// ---- POUs/UserPOUs/UserFunctions/ToRobotPoseSimple.TcPOU
FUNCTION ToRobotPoseSimple
VAR_INPUT
	x, y, theta : LREAL;
END_VAR
VAR
END_VAR
VAR_OUTPUT
	RobotPose : RobotPoseSimple;
END_VAR

RobotPose.x := x;
RobotPose.y := y;
RobotPose.theta := theta;

END_FUNCTION

// ---- POUs/UserPOUs/TrajectoryControl.TcPOU
//TrajectoryControl:
//GW2 side of the interface to GW3
FUNCTION_BLOCK TrajectoryControl
VAR_INPUT
	//interface to GW3
	// INPUTS to GW3
	xBoEnable AT%Q*: BOOL := FALSE;							// Freigabesignal für Fahrt, Roboter stoppt bei FALSE
	waypointList AT%Q*: ARRAY[0..100] OF RobotPoseSimple;	// Wegpunktliste mit Roboter-Posen in globalen Koordinaten (x, y, theta)
	newWaypointListAvailable AT%Q*: BOOL := FALSE;			// Status-Bit zur Signalisierung einer neuen WP-Liste
	xBoReset  AT%Q*: BOOL := FALSE;							
END_VAR
VAR_OUTPUT
	// OUTPUTS from GW3		
	yBoArrivedAtDestination AT%I*: BOOL 			:= FALSE;	// TRUE, wenn Ziel erreicht, Ziel entspricht letzten gültigen WP
	yUintWaypointIndex  	AT%I*: INT 				:= 0;		// COUNTER zur Anzeige, des Indexes des nächstes WP
	yRPposition 			AT%I*: RobotPoseSimple;				// aktuelle Roboterposition, für Simulationszwecke;
	yControllerState   	 	AT%I*: ControllerState;
	yVworldRef				AT%I*: RobotPoseSimple;
END_VAR

METHOD setWaypointList : BOOL
VAR_INPUT
	newWaypointList : ARRAY [0..100] OF RobotPoseSimple;
END_VAR
waypointList := newWaypointList;
END_METHOD

END_FUNCTION_BLOCK

// ---- POUs/UserPOUs/UserFunctions/ZEROS_RobotPoseSimple.TcPOU
FUNCTION ZEROS_RobotPoseSimple : Array[0..100] OF RobotPoseSimple
VAR_IN_OUT
	arr: ARRAY [0..100] OF RobotPoseSimple;
END_VAR
VAR
	i: INT;
END_VAR

FOR i := 0 TO 100 BY 1 DO
	arr[i] := ToRobotPoseSimple(x := 0, y := 0, theta := 0);
END_FOR

END_FUNCTION

// ---- POUs/UserPOUs/GW2/DS_GW1.TcPOU
PROGRAM DS_GW1
VAR
// Identifikation des Roboters
    //Robot_Number	AT%I*	: INT;	

// Local Variables for Mqtt Client handling
	fbIotMqttClient : FB_IotMqttClient;
	//ClientId : STRING(255);
    //ClientId : STRING(255) := CONCAT('HAWino_', INT_TO_STRING(.Var_HAWIno.Robot_Number));
	bSetParameter 	: BOOL := TRUE;
	bConnect 		: BOOL := TRUE;	
	
// Publish message
	initMQTT : BOOL := FALSE;
	sTopicPubToPowerMgmt : STRING(255); //:= CONCAT('Robots/PowerMgmt/Robot_', INT_TO_STRING(.Var_HAWIno.Robot_Number)); 	// ToDo: Bisher ist die Nummer des HAWino fest kodiert
	sTopicPubToPowerMgmt_SOC : STRING(255);// := CONCAT('Robots/PowerMgmt/SoC_Robot_', INT_TO_STRING(.Var_HAWIno.Robot_Number)); 
	sPayloadPub : STRING(2000);
	sPayloadPub1 : STRING(2000);		
	fbTimerPub 	: TON := (PT:=T#500MS);									// Intervall für das Senden des Akku-Status
	
//Received message
	bSubscribed    : BOOL;
	sTopicSubToPowerMgmt : STRING(255);// := CONCAT('PowerMgmt/Robots/Robot_', INT_TO_STRING(.Var_HAWIno.Robot_Number));	// ToDo: Bisher ist die Nummer des HAWino fest kodiert
	sTopicRcv      : STRING(255);
	sPayloadRcv    : STRING(255);
	fbMessageQueue : FB_IotMqttMessageQueue;
    fbMessage      : FB_IotMqttMessage;
	hrErrorOccurred : HRESULT; 			// Enthlt dern letzten augetretenen Fehler
	
	//wir geändert
	//sTopicSubToGW1: STRING(255);
	
// Variables for JSON
	fbJson			: FB_JsonSaxWriter;
	fbJsonDataType 	: FB_JsonReadWriteDataType;
	sJsonDoc       	: STRING(2000); 
	
// Local Variables for TwinCAT IoT Communication (TF6701) with direct link to EK1200 and TcCom
	//stMqtt_HAWino_In	AT%I*	: ST_PwrMgmt_HAWino_In;		// Attention! Don't link TIME Variables, otherwise we get an error!
	//stMqtt_HAWino_Out	AT%Q*	: ST_PwrMgmt_HAWino_Out;
	
	stMqtt_HAWino_In	 AT%I*: ST_PwrMgmt_HAWino_In;		// Attention! Don't link TIME Variables, otherwise we get an error!
	stMqtt_HAWino_Out	 AT%Q*: ST_PwrMgmt_HAWino_Out;
	
	SOC_Out : STRING(255);
	nBatteryTemperature	AT%I*	: INT;
	
	bComCheckAnswer	AT%Q*	: BOOL;
	
	stMqtt_HAWinoValues	: ST_PwrMgmt_HAWino;
	
	
// Timer to create a time stamp
	fbTimerTimestamp : TON := (PT:=T#71582M47S295MS);
	
// Local Vaiables to evaluate and act to input
	fbComCheckFlag	: RS;
	
	
	
	sTopicSubToFleetMgmt: STRING;
	Reset1: BOOL;
	//Input synccheck. robotdata has been read and can be used.
	txtReadInit AT%I* : BOOL := FALSE;
	
	// eigene Variablen	
	feedback: ARRAY[0..7] OF STRING := ['Verfügbar', 'Auftrag angenommen', 'Auf Anfahrt', 'Teil aufgenommen', 
											'Abmeldung', 'Auf Transport', 'Anmeldung', 'Teil abgelegt'];
	sTopicPubToGW1: STRING(255) := CONCAT('VPJ/Robot_', INT_TO_STRING(.Var_HAWIno.Robot_Number));
	s0: BOOL := 1;
	s1, s2, s3, s4, s5, s6, s7: BOOL := 0;
	AuftragDa: BOOL;
	Timer1 : TON;
	Timer2 : TON;
	startTime1: BOOL;
	startTime2: BOOL;
	WerkstueckAusgelesen: BOOL;
	i: INT := 0;

END_VAR

//Dummy Programm als Schnittstelle für Gewerk 1

//Case machen! preop op
txtReadInit := MQTT.txtReadInit;
IF txtReadInit THEN
	IF NOT initMQTT THEN
		sTopicPubToPowerMgmt  := CONCAT('Robots/PowerMgmt/Robot_', INT_TO_STRING(.Var_HAWIno.Robot_Number)); 	
		sTopicPubToPowerMgmt_SOC  := CONCAT('Robots/PowerMgmt/SoC_Robot_', INT_TO_STRING(.Var_HAWIno.Robot_Number)); 
		sTopicSubToPowerMgmt  := CONCAT('PowerMgmt/Robots/Robot_', INT_TO_STRING(.Var_HAWIno.Robot_Number));
		//sTopicSubToGW1  := CONCAT('VPJ/Robot_', INT_TO_STRING(.Var_HAWIno.Robot_Number));
		initMQTT:= TRUE;
	END_IF
	
	stMqtt_HAWinoValues.Output.nRobotNumber := .Var_HAWIno.Robot_Number;			// Anpassen für jeden HAWino
	
	fbTimerTimestamp(In:= NOT fbTimerTimestamp.Q, ET=>stMqtt_HAWinoValues.Output.tTimestamp);
	
	stMqtt_HAWinoValues.Output.fSoC := stMqtt_HAWino_In.fSoC;
	
	stMqtt_HAWinoValues.Output.fActualBatteryCurrent := stMqtt_HAWino_In.fActualBatteryCurrent;
	stMqtt_HAWinoValues.Output.fActualBatteryVoltage := stMqtt_HAWino_In.fActualBatteryVoltage;
	
	//stMqtt_HAWinoValues.Output.fActualBatteryCurrent := stMqtt_HAWino_In.fActualBatteryCurrent;
	//stMqtt_HAWinoValues.Output.fActualBatteryVoltage := stMqtt_HAWino_In.fActualBatteryVoltage;
	
	
	
	
	// Skalierung der Temperaturwerte des Akkus
	stMqtt_HAWinoValues.Output.fBatteryTemperature := FKT_Scale(Rohwert := nBatteryTemperature, 
																	X1 := -500,
																	X2 := 1500, 
																	Y1 := -50,
																	Y2 := 150);
																	
	// Ausgabe der erwarteten Laufzeit des Roboters
	stMqtt_HAWinoValues.Output.nEstimatedRunningTime	:= LIMIT(0,stMqtt_HAWino_In.nEstimatedRunningTime,172800);		// Max. 48 Stunden sollen dargestellt werden
	stMqtt_HAWinoValues.Output.nEstimatedChargingTime	:= LIMIT(0,stMqtt_HAWino_In.nEstimatedChargingTime,172800);		// Max. 48 Stunden sollen dargestellt werden
	
	
	// Antworten auf den Kommunikationstest und des Ladetests
	stMqtt_HAWinoValues.Output.bCheckCurrentDetected := stMqtt_HAWino_In.bCheckCurrentDetected;
	stMqtt_HAWinoValues.Output.bComCheckAnswer := stMqtt_HAWino_In.bComCheckAnswer;
	
	
			
	
	
	
	
	//
	// Setting the parameters for establishing the connection to the Mqtt Broker and initializing the connection.
	//
	IF bSetParameter THEN
		fbIotMqttClient.sHostName := '192.168.0.11';	// IP-Adresse des Servers
		fbIotMqttClient.nHostPort := 1883;
		//fbIotMqttClient.sClientId := ClientId;
		fbIotMqttClient.sClientId := CONCAT('Robot_', INT_TO_STRING(.Var_HAWIno.Robot_Number));
		fbIotMqttClient.sTopicPrefix := '';
		//fbIotMqttClient.nKeepAlive:= 60; 
		fbIotMqttClient.sUserName:= 'VPJ';
		fbIotMqttClient.sUserPassword:= 'R462';
		//fbIotMqttClient.stWill:= ; 
		//fbIotMqttClient.stTLS:= ;
		fbIotMqttClient.ipMessageQueue := fbMessageQueue;
	
		bSetParameter := FALSE;
	END_IF
	
	
	//
	// This method -> MUST BE CALLED CYCLICALLY <- to ensure background communication with the MQTT broker.
	//
	fbIotMqttClient.Execute(bConnect);
	
	IF fbIotMqttClient.bError THEN
		// ToDo: add error logging here
		hrErrorOccurred := fbIotMqttClient.hrErrorCode;
	END_IF
	
		
	IF fbIotMqttClient.bConnected THEN		// Kontrolle, ob der Broker verbunden ist
		IF NOT bSubscribed THEN
			//
			// Abbonieren der Toopics, welche vom PowerMgmt kommen
			//
			bSubscribed := fbIotMqttClient.Subscribe(sTopic:=sTopicSubToPowerMgmt, eQoS:=TcIotMqttQos.AtMostOnceDelivery);
			IF fbIotMqttClient.bError THEN
				// ToDo: add my error logging here
				hrErrorOccurred := fbIotMqttClient.hrErrorCode;
			END_IF
			
			//
			// Abbonieren der Toopics, welche vom Gewerk 1 kommen
			//
			//Abbonieren von Topic: VPJ/Roboter
			//bSubscribed := fbIotMqttClient.Subscribe(sTopic:=sTopicSubToGW1, eQoS:=TcIotMqttQos.AtMostOnceDelivery);
			
			
			//bSubscribed := fbIotMqttClient.Subscribe(sTopic:=sTopicSubToFleetMgmt, eQoS:=TcIotMqttQos.AtMostOnceDelivery);
			//IF fbIotMqttClient.bError THEN
				// ToDo: add my error logging here
			//	hrErrorOccurred := fbIotMqttClient.hrErrorCode;
			//END_IF
			
		END_IF
	END_IF	
	
	
	
	// Senden der MQTT- Nachrichten
	
	
	IF fbIotMqttClient.bConnected THEN			// Kontrolle, ob Broker verbunden ist
		fbTimerPub(IN:=TRUE);
		
		//
		// publish new paylod every 500 MS
		//
		IF fbTimerPub.Q THEN					// Abwarten des oben eingestellten Intervalls
			fbTimerPub(IN:=FALSE);
			
			//
			// Nachricht an PowerMgmt
			//
			fbJson.ResetDocument();
			fbJsonDataType.AddJsonValueFromSymbol(fbJson, 'ST_PwrMgmt_HAWino_In', SIZEOF(stMqtt_HAWinoValues.Output), ADR(stMqtt_HAWinoValues.Output));
			//sJsonDoc := fbJson.GetDocument();
			fbJson.CopyDocument(sJsonDoc, SIZEOF(sJsonDoc));
			
			sPayloadPub := sJsonDoc;	
			fbIotMqttClient.Publish(sTopic:= sTopicPubToPowerMgmt, 
										pPayload:= ADR(sPayloadPub), 
										nPayloadSize:= LEN2(ADR(sPayloadPub))+1, 										
										eQoS:= TcIotMqttQos.AtMostOnceDelivery, 
										bRetain:= FALSE, 
										bQueue:= FALSE);
									
			
			SOC_Out	:= CONCAT( '{"SoC" : ',LREAL_TO_STRING(stMqtt_HAWinoValues.Output.fSoC));
			SOC_Out	:= CONCAT( SOC_Out,'}');
			
			
			
			
			//SOC_Out := 	LREAL_TO_STRING(stMqtt_HAWinoValues.Output.fSoC);
			
						
			fbIotMqttClient.Publish(sTopic:= sTopicPubToPowerMgmt_SOC, 
										pPayload:=ADR(SOC_Out), 
										nPayloadSize:= INT_TO_UDINT(LEN(SOC_Out)),
										eQoS:= TcIotMqttQos.AtMostOnceDelivery, 
										bRetain:= FALSE, 
										bQueue:= FALSE);
										
										
			IF fbIotMqttClient.bError THEN
				// ToDo: add error logging here
				hrErrorOccurred := fbIotMqttClient.hrErrorCode;
			END_IF	
			
			//
			// ...
			//	
			//
			// Nachricht an GW1 - Produktionsauftrag
			//
			//Statemaschine
			Timer1(IN:= startTime1, PT:=T#10S);
			Timer2(IN:= startTime2, PT:=T#10S);
	
			//Rückmeldung Verfügbar
			sPayloadPub1 := CONCAT( '{"status" : ', feedback[i]);
			sPayloadPub1 := CONCAT( sPayloadPub1,'}');
			
			fbIotMqttClient.Publish(sTopic:= sTopicPubToGW1, 
											pPayload:=ADR(sPayloadPub1), 
											nPayloadSize:= INT_TO_UDINT(LEN(sPayloadPub1)),
											eQoS:= TcIotMqttQos.AtMostOnceDelivery, 
											bRetain:= FALSE, 
											bQueue:= FALSE);
											
			i := 2;
											
			//Warten auf Auftrag
			IF s0 AND NOT s1 AND AuftragDa THEN
				s0 := 0; s1 := 1;
				//Rückmeldung Auftrag angenommen
				i := 1;
				//fbIotMqttClient.Publish(sTopic:= sTopicPubToGW1, 
											//pPayload:=ADR(feedback[1]), 
											//nPayloadSize:= INT_TO_UDINT(LEN(feedback[1])),
											//eQoS:= TcIotMqttQos.AtMostOnceDelivery, 
											//bRetain:= FALSE, 
											//bQueue:= FALSE);
				startTime1 := 1;
			END_IF
			IF s1 AND NOT s2 AND Timer1.Q THEN
				startTime1 := 0;
				s1 := 0; s2 := 1;
				//Rückmeldung Auf Anfahrt
				i := 2;
				//fbIotMqttClient.Publish(sTopic:= sTopicPubToGW1, 
											//pPayload:=ADR(feedback[2]), 
											//nPayloadSize:= INT_TO_UDINT(LEN(feedback[2])),
											//eQoS:= TcIotMqttQos.AtMostOnceDelivery, 
											//bRetain:= FALSE, 
											//bQueue:= FALSE);
				startTime2 := 1;
			END_IF
			IF s2 AND NOT s3 AND Timer2.Q THEN
				startTime2 := 0;
				s2 := 0; s3 := 1;
				//Rückmeldung Teil aufgenommen
				i := 3;
				fbIotMqttClient.Publish(sTopic:= sTopicPubToGW1, 
											pPayload:=ADR(feedback[3]), 
											nPayloadSize:= INT_TO_UDINT(LEN(feedback[3])),
											eQoS:= TcIotMqttQos.AtMostOnceDelivery, 
											bRetain:= FALSE, 
											bQueue:= FALSE);
				startTime1 := 1;
			END_IF
			IF s3 AND NOT s4 AND Timer1.Q THEN
				startTime1 := 0;
				s3 := 0; s4 := 1;
				//Rückmeldung Abmeldung
				i := 4;
				//fbIotMqttClient.Publish(sTopic:= sTopicPubToGW1, 
											//pPayload:=ADR(feedback[4]), 
											//nPayloadSize:= INT_TO_UDINT(LEN(feedback[4])),
											//eQoS:= TcIotMqttQos.AtMostOnceDelivery, 
											//bRetain:= FALSE, 
											//bQueue:= FALSE);
			END_IF
			//Warten auf Werkstück ausgelesen
			IF s4 AND NOT s5 AND WerkstueckAusgelesen THEN
				s4 := 0; s5 := 1;
				//Rückmeldung Auf Transport
				fbIotMqttClient.Publish(sTopic:= sTopicPubToGW1, 
											pPayload:=ADR(feedback[5]), 
											nPayloadSize:= INT_TO_UDINT(LEN(feedback[5])),
											eQoS:= TcIotMqttQos.AtMostOnceDelivery, 
											bRetain:= FALSE, 
											bQueue:= FALSE);
				startTime2 := 1;
			END_IF
			IF s5 AND NOT s6 AND Timer2.Q THEN
				startTime2 := 0;
				s2 := 0; s3 := 1;
				//Rückmeldung Anmeldung
				fbIotMqttClient.Publish(sTopic:= sTopicPubToGW1, 
											pPayload:=ADR(feedback[6]), 
											nPayloadSize:= INT_TO_UDINT(LEN(feedback[6])),
											eQoS:= TcIotMqttQos.AtMostOnceDelivery, 
											bRetain:= FALSE, 
											bQueue:= FALSE);
			END_IF
			//Warten auf Werkstück ausgelesen
			IF s6 AND NOT s7 AND WerkstueckAusgelesen THEN
				s6 := 0; s7 := 1;
				//Rückmeldung Teil abgelegt
				fbIotMqttClient.Publish(sTopic:= sTopicPubToGW1, 
											pPayload:=ADR(feedback[7]), 
											nPayloadSize:= INT_TO_UDINT(LEN(feedback[7])),
											eQoS:= TcIotMqttQos.AtMostOnceDelivery, 
											bRetain:= FALSE, 
											bQueue:= FALSE);
				startTime1 := 1;
			END_IF
			IF s7 AND NOT s0 AND Timer1.Q THEN
				startTime1 := 0;
				s7 := 0; s0 := 1;
				//Rückmeldung Verfügbar
				fbIotMqttClient.Publish(sTopic:= sTopicPubToGW1, 
											pPayload:=ADR(feedback[0]), 
											nPayloadSize:= INT_TO_UDINT(LEN(feedback[0])),
											eQoS:= TcIotMqttQos.AtMostOnceDelivery, 
											bRetain:= FALSE, 
											bQueue:= FALSE);
			END_IF
			
	//Hier müsste noch die ankommenden Daten vom GW1 ausglesen und ausgewertet (AuftragDa und WerkstueckAusgelesen schreiben) werden
	//IN MQTT könnte dann evtl das Auslesen/Subscribe wegfallen fürs erste...


		END_IF
	END_IF
	
	
	
	// Verarbeiten der Subscriptions
	
	
	IF fbMessageQueue.nQueuedMessages > 0 THEN			// Kontrolle, ob neue Daten vorliegen
		IF fbMessageQueue.Dequeue(fbMessage:=fbMessage) THEN
			fbMessage.GetTopic(pTopic:=ADR(sTopicRcv), nTopicSize:=SIZEOF(sTopicRcv) );
			fbMessage.GetPayload(pPayload:=ADR(sPayloadRcv), nPayloadSize:=SIZEOF(sPayloadRcv), bSetNullTermination:=FALSE);
				
			//
			// Message from PowerMgmt
			//
			IF fbMessage.CompareTopic(sTopic:=sTopicSubToPowerMgmt) THEN		// Wenn die Daten vom PowerMgmt kommen, dann führe folgenede Aktion aus
				
			// Json-String aufteilen und in Variablen schreiben
				fbJsonDataType.SetSymbolFromJson(sPayloadRcv,'ST_PwrMgmt_HAWino_Out',SIZEOF(stMqtt_HAWinoValues.Input),ADR(stMqtt_HAWinoValues.Input));
			END_IF
		
			//
			// Hier werden weitere Topics verarbeitet
			//
			
		END_IF
	END_IF		
	
	
	
	
	// Evaulierung der empfangenen Daten
	
	//
	// ToDo: Plausibilitätsprüfung von stMqtt_HAWinoValues.Input und evt. TypConversion
	// Attention! The assignment of input to output is correct. Don `t change!
	//	
	
	stMqtt_HAWino_Out.bChargingActive := stMqtt_HAWinoValues.Input.bChargingActive;
	stMqtt_HAWino_Out.bExternalRecalibrationTrigger := stMqtt_HAWinoValues.Input.bExternalRecalibrationTrigger;
	stMqtt_HAWino_Out.fExternalRecalibrationValue := stMqtt_HAWinoValues.Input.fExternalRecalibrationValue;
	
	
	// Hier Communication Check einbauen
	
	//fbComCheckFlag(Set:= stMqtt_HAWinoValues.Input.bComCheckRequest, 
	//					Reset1:= NOT stMqtt_HAWinoValues.Input.bComCheckRequest,
	//					Q1 => bComCheckAnswer);
	bComCheckAnswer	:= TRUE;
					
END_IF

END_PROGRAM

// ---- POUs/UserPOUs/GW3ControlAlgorithm/NonLinearController.TcPOU
FUNCTION_BLOCK NonlinearController
VAR_INPUT
	robotPose				: RobotPoseSimple;		// Actual robot pose [x, y, theta] in global frame
	robotPoseRef			: RobotPoseSimple;		// Reference robot pose [x, y, theta] in global frame
	robotVelocitiesRef		: RobotPoseSimple;		// Reference robot velocites [vX, vY, omega] in global frame
	vRef					: LREAL;				// Reference linear velocity along path
	enable					: BOOL;
END_VAR

VAR_OUTPUT
	vX						: LREAL;				// Output reference x-velocity in global frame for low-level controller
	vY						: LREAL;				// Output reference y-velocity in global frame for low-level controller
	omega					: LREAL;				// Output refernce angular velocity for low-level controller
	reachedReference		: BOOL;
END_VAR

VAR
	k1, k2, k3				: LREAL;				// Control parameters
	xE, yE, thetaE			: LREAL;				// Robot pose error
	u1, u2					: LREAL;				// Control variables
	xRef, yRef, thetaRef	: LREAL;				// 
	omegaRef				: LREAL;				//
	xAct, yAct, thetaAct	: LREAL;	
	vTransMax				: LREAL := 0.93;
	vRotMax					: LREAL := 1.57;
	positionTolerance		: LREAL := 0.002;
	orientationTolerance	: LREAL := 0.01;
	vRef					: LREAL;				// Reference linear velocity along path
END_VAR

// Reset effective control varibales
vX := 0;
vY := 0;
omega := 0;

k1 := 10;
k3 := 1;

IF enable THEN
	xRef := robotPoseRef.x / 1000;
	yRef := robotPoseRef.y / 1000;
	thetaRef := robotPoseRef.theta;
	omegaRef := robotVelocitiesRef.theta;
	xAct := robotPose.x / 1000;
	yAct := robotPose.y / 1000;
	thetaAct := robotPose.theta;
	
	vRef := SQRT(EXPT(xRef, 2) + EXPT(yRef, 2));

	// Suggested value for k2
	k2 := 2 * ABS(vRef) * SQRT(k3);
	
	// Control errors in mobile reference frame
	xE := COS(thetaAct) * (xRef - xAct) + SIN(thetaAct) * (yRef - yAct);
	yE := -SIN(thetaAct) * (xRef - xAct) + COS(thetaAct) * (yRef - yAct);
	thetaE := -(thetaRef - thetaAct);
	
	// Control law
	u2 := -k2 * thetaE + k3 * vRef * yE * SI(thetaE);
	u1 := vRef * (COS(thetaE) - 1) + yE * (omegaRef + u2) + k1 * xE;
	
	// Write effective control variables
	vX := (u1 + vRef) * COS(thetaAct);
	vY := (u1 + vRef) * SIN(thetaAct);
	omega := u2 + omegaRef;
	
	// Limit effective control variables
	IF (vX > vTransMax) THEN
		vX := vTransMax;
	ELSIF (vX < - vTransMax) THEN
		vX := - vTransMax;
	END_IF
	
	IF (vY > vTransMax) THEN
		vY := vTransMax;
	ELSIF (vY < - vTransMax) THEN
		vY := - vTransMax;
	END_IF
	
	IF (omega > vRotMax) THEN
		omega := vRotMax;
	ELSIF (omega < - vRotMax) THEN
		omega := - vRotMax;
	END_IF
	
	reachedReference := (SQRT(EXPT(xE, 2) + EXPT(yE, 2)) < positionTolerance) AND (ABS(thetaE) < orientationTolerance);
	
	// Scale back to mm / s
	vX := vX * 1000;
	vY := vY * 1000;
END_IF

METHOD reset : BOOL
VAR_INPUT
END_VAR
reachedReference := FALSE;
END_METHOD

END_FUNCTION_BLOCK

// ---- POUs/UserPOUs/UserFunctions/SI.TcPOU
FUNCTION SI : LREAL
VAR_INPUT
	x	: LREAL;
END_VAR
VAR
END_VAR

IF (x > -0.001) AND (X < 0.001) THEN 
	SI := 1.0;
ELSE
	SI := SIN(x) / x;
END_IF

END_FUNCTION

// ---- POUs/UserPOUs/GW3ControlAlgorithm/SimpleObserver.TcPOU
//SimpleObserver:
//Implements a simple observer which assumes the camera position is the true position of the robot whenever camera data arrives. Between new cam data
//odometry is used to correct the robots position. The cameras latency is also considered by correcting the arrived camera data with odometry based correction
//within the time interval of the latency. The observer is implemented in Simulink and is linked within this FB to abstract the implementation of the observer from the
//main control algorithm. Inside the Simulink model all coordinates are considered as world coordinates, following that the transformation of between robot and world coordinates 
//is implemented in ST.
FUNCTION_BLOCK SimpleObserver
VAR_INPUT
	xCameraPose:	RobotPoseSimple;
	xVxRobot: 		LREAL;
	xVyRobot: 		LREAL;
	xOmegaRobot: 	LREAL;
	theta:			LREAL; //theta for I/O Lineraztion only explicitly Input for FF-Linearization
END_VAR

VAR_OUTPUT
	yObserverdPose: 	RobotPoseSimple;
END_VAR

VAR
	newCamDataArrived: BOOL;
	camDataOld, observerError, observedPosition, vWorld: RobotPoseSimple;
	pulseGenerator: TP;
	
	delayedCycles		AT%Q* 	: INT	:= 20;
	delayedPosition: ARRAY [0..140] OF RobotPoseSimple;
	
	
	K : ARRAY [0..2,0..2] OF LREAL 		:= [25, 0 ,0,
									  		0, 25, 0,
									  		0, 0, 25];
END_VAR

//transform roboter velocities into world velocities and pass them to Simulink
Robot2World( 
	vx_robot 	:= xVxRobot,
	vy_robot 	:= xVyRobot,
	omega_robot := xOmegaRobot,
	theta		:= yObserverdPose.theta,
	vx_world 	=> vWorld.x,
	vy_world  	=> vWorld.y,
	omega_world => vWorld.theta);
	
checkForNewCameraData();

//systime(START:=newCamDataArrived);	// TEST

delayPosition();
//if cam data arrived correct
IF newCamDataArrived THEN
	//calculate observer error
	observerError := SubtractRPS(xCameraPose,delayedPosition[delayedCycles]);
	//do the feedback correction
	observedPosition := AddRPS(observedPosition, ScaleRPS(c := Var_HAWIno.CONTROLLER_CYCLE_TIME, AddRPS(vWorld, MatrixTimesRPS(K, observerError))));
ELSE
	observedPosition := AddRPS(observedPosition, ScaleRPS(c := Var_HAWIno.CONTROLLER_CYCLE_TIME, vWorld));
END_IF


//set Outputs
yObserverdPose 	:= observedPosition;
camDataOld 		:= xCameraPose;

METHOD checkForNewCameraData : BOOL
VAR_INPUT
END_VAR
newCamDataArrived := (camDataOld.x <> xCameraPose.x OR camDataOld.y <> xCameraPose.y OR camDataOld.theta <> xCameraPose.theta) //cahnge in one of the positions
					 AND xCameraPose.x <> 0 AND xCameraPose.y <> 0;		//valid data
END_METHOD

METHOD PRIVATE delayPosition : BOOL
VAR_INPUT
END_VAR
VAR
	i: INT := 0;
END_VAR
FOR i := 0 TO delayedCycles-1 DO
	delayedPosition[i+1] := delayedPosition[i];
END_FOR
delayedPosition[0] := observedPosition;
END_METHOD

METHOD reset : BOOL
VAR_INPUT
END_VAR
VAR
	
END_VAR
reset := FALSE;
IF newCamDataArrived THEN
	observedPosition := xCameraPose;
	reset := TRUE;
END_IF
END_METHOD

END_FUNCTION_BLOCK

// ---- POUs/UserPOUs/UserFunctions/MatrixTimesRPS.TcPOU
FUNCTION MatrixTimesRPS : RobotPoseSimple
VAR_INPUT
	K: ARRAY [0..2,0..2] OF LREAL;
	pose: RobotPoseSimple;
END_VAR

//2.) apply gain on errors
MatrixTimesRPS.x 	 := K[0,0] * pose.x + K[1,0] * pose.y + K[2,0] * pose.theta;
MatrixTimesRPS.y 	 := K[0,1] * pose.x + K[1,1] * pose.y + K[2,1] * pose.theta;
MatrixTimesRPS.theta := K[0,2] * pose.x + K[1,2] * pose.y + K[2,2] * pose.theta;

END_FUNCTION

// ---- POUs/UserPOUs/GW3ControlAlgorithm/SimpleTrajectory.TcPOU
//SimpleTrajectory:
//implements a simple trajectory which takes a waypoint list od max 100 poses. The points are outputted one by one as reference pose with no further modifications.
//The trajectory switches to the next pose if the x-y-distance d between  'currentPose' and the current reference 'referencePose[WPLidx]'
//is within a tolerance 'tol' to the current .
//waypoint. If all three coordinates of the waypoint are set to -1 the trajectory marks itself
//as finished.
FUNCTION_BLOCK SimpleTrajectory
VAR_INPUT
	currentPose			: RobotPoseSimple; 
END_VAR
VAR_OUTPUT
	finished			: BOOL 				:= FALSE;
	referencePose		: RobotPoseSimple;
	WPLidx 				: INT 				:= 0;
END_VAR
VAR
	wayPointList		: ARRAY [0..100] OF RobotPoseSimple;
	dPosition: LREAL  := 0;
	dOrientation:   LREAL  := 0;
	tolPosition: LREAL := 10; 
	tolOrientation: LREAL := 0.314/2;
END_VAR

//calculte current distance from reference point
dPosition := SQRT(EXPT(currentPose.x - wayPointList[WPLidx].x, 2) + EXPT(currentPose.y - wayPointList[WPLidx].y,2));
dOrientation := ABS(currentPose.theta - wayPointList[WPLidx].theta);

IF dOrientation < tolOrientation AND dPosition < tolPosition AND NOT finished AND WPLidx < 100 THEN
	WPLidx := WPLidx +1;
END_IF
IF wayPointList[WPLidx].x = -1 AND wayPointList[WPLidx].y = -1 AND wayPointList[WPLidx].theta = -1 THEN
	finished := TRUE;
END_IF
referencePose := wayPointList[WPLidx];

METHOD setRobotPose : RobotPoseSimple
VAR_INPUT
	newPose: RobotPoseSimple;
END_VAR
setRobotPose := newPose;
END_METHOD

METHOD setWaypointList : ARRAY [0..100] OF RobotPoseSimple
VAR_INPUT
	newWayPointList	: ARRAY [0..100]  OF RobotPoseSimple;
END_VAR
WPLidx 			:= 0; 						//reset
finished 		:= FALSE;
wayPointList 	:= newWayPointList;
END_METHOD

END_FUNCTION_BLOCK

// ---- POUs/UserPOUs/GW3PathAndTrajectoryPlanning/LinearCurve.TcPOU
(*Class: Linear Curve
Implementation of a linear Curve. The linear Spline is defined uniquely by two waypoints.
*)
FUNCTION_BLOCK LinearCurve EXTENDS Curve
VAR_INPUT
	wayPoints: ARRAY[0..1] OF RobotPoseSimple; //Input waypoints for creation of the linear Spline. First element should be startPoint and 
END_VAR
VAR_OUTPUT
END_VAR
VAR
	init : BOOL := FALSE;
END_VAR

startPoint := wayPoints[0];
endPoint   := wayPoints[1];

startPoint.theta	:= ATAN2(endPoint.y-startPoint.y, endPoint.x-startPoint.x); 
endPoint.theta		:= startPoint.theta;
lengthVar 			:= calculateLength();

(* 
Implementation of abstract Spline method.
For internal inital length calculation, should be called in the constructor => protected
*)
METHOD PROTECTED  calculateLength : LREAL
VAR_INPUT
END_VAR
calculateLength := SQRT(EXPT(startPoint.x - endPoint.x,2) + EXPT(startPoint.y - endPoint.y, 2));
END_METHOD

(* 
Implementation of abstract Spline method.
Calculates the derivate of the spline at an arbitrary arcLength. Should be implmented for order one and two. Invalid 
orders should write a -1 in every component of the return value.
*)
METHOD  diff : RobotPoseSimple
VAR_INPUT
	arcLength: LREAL; //arcLength at which the corresponding derivative should be calculated
	order: INT := 1;  //optional: order of the derivate, should be implemented for 1 and 2, default: 1
END_VAR
IF order = 1 THEN
	diff.x 		:= COS(startPoint.theta);
	diff.y 		:= SIN(startPoint.theta);
	diff.theta   := -1; //not used
ELSIF order = 2 THEN
	diff.x 		:= 0;
	diff.y 		:= 0;
	diff.theta   := -1; //not used
ELSE
	//invalid input
	diff.x 		:= -1; 
	diff.y 		:= -1;
	diff.theta   := -1; //not used
END_IF
END_METHOD

(*
Implementation of abstract Spline method.
Gets the configuration of the Spline at any given arcLength. 
*)
METHOD getPoint : RobotPoseSimple
VAR_INPUT
	arcLength	: LREAL;
END_VAR
getPoint.x		:= COS(startPoint.theta)*arcLength + startPoint.x;
getPoint.y		:= SIN(startPoint.theta)*arcLength + startPoint.y;
getPoint.theta  := -1; //not used
END_METHOD

END_FUNCTION_BLOCK

// ---- POUs/UserPOUs/UserFunctions/ArrayToStruct.TcPOU
FUNCTION ArrayToStruct : ARRAY[1..100]  OF RobotPoseSimple 
VAR_INPUT
	x: ARRAY [1..10] OF LREAL;
	y: ARRAY [1..10] OF LREAL;
	theta: LREAL;
END_VAR
VAR
	i: INT := 1;
	lastPosition: INT := 1;
END_VAR
VAR_OUTPUT
	outputArray: ARRAY[1..100]  OF RobotPoseSimple;
END_VAR

//FOR i := 0 TO 100 BY 1 DO
	//IF x[i] <> -1.0 THEN //nicht -1 oder ende des Arrays
		//outputArray[i].x := x[i];
		//outputArray[i].y := y[i];
		//outputArray[i].theta := -1;
		//lastPosition := i;
	//ELSE
		//outputArray[i].x := -1;
		//outputArray[i].y := -1;	
	//END_IF;
//END_FOR;

//outputArray[lastPosition].theta := theta;

END_FUNCTION

// ---- POUs/UserPOUs/UserFunctions/calcTimeDiff.TcPOU
FUNCTION calcTimeDiff : LREAL
VAR_INPUT
	TimeCam : TIMESTRUCT;
	TimeSys : TIMESTRUCT; 
END_VAR
VAR
END_VAR

END_FUNCTION

// ---- POUs/UserPOUs/UserFunctions/RPS2ARRAY.TcPOU
//Converts a RobotPoseSimple to a ARRAY [0..2] OF LREAL
FUNCTION RPS2ARRAY : ARRAY [0..2] OF LREAL
VAR_INPUT
	pose: RobotPoseSimple;
END_VAR
VAR
END_VAR

RPS2ARRAY[0] := pose.x;
RPS2ARRAY[1] := pose.y;
RPS2ARRAY[2] := pose.theta;

END_FUNCTION

// ---- POUs/UserPOUs/UserFunctions/RP2ARRAY.TcPOU
//converts a RobotPose into a ARRAY [0..3] OF LREAL
FUNCTION RP2ARRAY : ARRAY [0..3] OF LREAL
VAR_INPUT
	pose: RobotPose;
END_VAR
VAR
END_VAR

RP2ARRAY[0] := pose.x;
RP2ARRAY[1] := pose.y;
RP2ARRAY[2] := pose.theta;
RP2ARRAY[3] := pose.e;

END_FUNCTION
